	rFlodesDifferensMellanMinOchMax : REAL;
	rFlodesHojning1 : REAL; // Flödeshöjning uträknat.
	rFlodesHojning2 : REAL; // Flödeshöjning uträknat.
	rFlodesHojning3 : REAL; // Flödeshöjning uträknat.
	rFlodesHojning4 : REAL; // Flödeshöjning uträknat.
	rFlodesHojning5 : REAL; // Flödeshöjning uträknat.
	rFlodesHojning6 : REAL; // Flödeshöjning uträknat.
	rFlodesHojning7 : REAL; // Flödeshöjning uträknat.
	rFlodesHojning8 : REAL; // Flödeshöjning uträknat.
	rFlodesHojning9 : REAL; // Flödeshöjning uträknat.
	rFlodesHojning10 : REAL; // Flödeshöjning uträknat.
	rFlodesHojning11 : REAL; // Flödeshöjning uträknat.
	rFlodesHojning12 : REAL; // Flödeshöjning uträknat.
	rFlodesHojning13: REAL; // Flödeshöjning uträknat.
	rFlodesHojning14 : REAL; // Flödeshöjning uträknat.
	rFlodesHojning15 : REAL; // Flödeshöjning uträknat.
	rOmraknadFlodeskompenseringsSignal1 : REAL; // Flödeskompenseringsinput omräknad till 0-100 värde.
	rOmraknadFlodeskompenseringsSignal2 : REAL; // Flödeskompenseringsinput omräknad till 0-100 värde.
	rOmraknadFlodeskompenseringsSignal3 : REAL; // Flödeskompenseringsinput omräknad till 0-100 värde.
	rOmraknadFlodeskompenseringsSignal4 : REAL; // Flödeskompenseringsinput omräknad till 0-100 värde.
	rOmraknadFlodeskompenseringsSignal5 : REAL; // Flödeskompenseringsinput omräknad till 0-100 värde.
	rOmraknadFlodeskompenseringsSignal6 : REAL; // Flödeskompenseringsinput omräknad till 0-100 värde.
	rOmraknadFlodeskompenseringsSignal7 : REAL; // Flödeskompenseringsinput omräknad till 0-100 värde.
	rOmraknadFlodeskompenseringsSignal8 : REAL; // Flödeskompenseringsinput omräknad till 0-100 värde.
	rOmraknadFlodeskompenseringsSignal9 : REAL; // Flödeskompenseringsinput omräknad till 0-100 värde.
	rOmraknadFlodeskompenseringsSignal10 : REAL; // Flödeskompenseringsinput omräknad till 0-100 värde.
	rOmraknadFlodeskompenseringsSignal11 : REAL; // Flödeskompenseringsinput omräknad till 0-100 värde.
	rOmraknadFlodeskompenseringsSignal12 : REAL; // Flödeskompenseringsinput omräknad till 0-100 värde.
	rOmraknadFlodeskompenseringsSignal13 : REAL; // Flödeskompenseringsinput omräknad till 0-100 värde.
	rOmraknadFlodeskompenseringsSignal14 : REAL; // Flödeskompenseringsinput omräknad till 0-100 värde.
	rOmraknadFlodeskompenseringsSignal15 : REAL; // Flödeskompenseringsinput omräknad till 0-100 värde.
	bSekvensFlagga : BOOL;
	wResetConfirmed : WORD;
	
	fbSetpointConfirmed : FB_MBReadRegs;
	fbWriteSetpoint: FB_MBWriteSingleReg;
	rFlowSetpoint : REAL;
	wFlowSetpoint : WORD;
	wFlowSetpointConfirmed : WORD;
	bExecute1 : BOOL;
	wFlow : WORD;
	wOperationPoint : WORD;
	
	fbDamperPosition : FB_MBReadRegs;

	
	fbProcessValue : FB_MBReadRegs;
			
	fbReadValues : FB_MBReadRegs;
	
	fbOperationModeConfirmed : FB_MBReadRegs;
	fbWriteOperationMode: FB_MBWriteSingleReg;
	wOperationModeConfirmed : WORD;
	
	fbModeConfirmed : FB_MBReadRegs;
	fbWriteMode: FB_MBWriteSingleReg;
	wModeConfirmed : WORD;
	
	bExecute2 : BOOL;
	bExecute3 : BOOL;
	bExecute4 : BOOL;

	fbDoubleControlledModbusHoldingMinFlow,fbDoubleControlledModbusHoldingMaxFlow: fbDoubleControlledModbusHolding;
	fbHoldingRead : FB_MBReadRegs;
	
	rTemp : REAL; 
	sIP: STRING(255);
	sPort: STRING(255);
	sModbusID: STRING(255);
	sModbusLoop: STRING(255);
	sTemp: STRING(255);
	
	wWtest : WORD;
	
	rMid : REAL;
	
	//Kommunikationsfel
	fbKommTof : tof; 
	fbKommTon : ton;
END_VAR
VAR_INPUT PERSISTENT
	M AT %M*  : BOOL; // Manuellt läge börvärde~wp:
	OPM AT %M*  : REAL; // Manuellt börvärde~wp:[unit]%[format]0
END_VAR

//Modbus konfiguering
	sIP := CONCAT (SIPAddr, '');
	sPort := CONCAT ('<br>Port: ', UINT_TO_STRING(nTCPPort)); 								
	sModbusID := CONCAT('<br>ID: ', UINT_TO_STRING(nUnitID));
	sModbusLoop := CONCAT('<br>Loop: ', INT_TO_STRING(nModbusLoop));
	sTemp := sIP;
	sTemp := CONCAT(sTemp, sPort);
	sTemp := CONCAT(sTemp, sModbusID);
	sTemp := CONCAT(sTemp, sModbusLoop);
	PV8 := sTemp;

	bSekvensFlagga := oaksGVL.aBModbusSekvens[nModbusLoop] = UINT_TO_INT(nUnitID);
	//fbTp01(IN:=oaksGVL.aBModbusSekvens[nModbusLoop] = UINT_TO_INT(nUnitID) , PT:=T#5S , Q=> , ET=> );
	
	rFlodesDifferensMellanMinOchMax := SP2 - SP1;
	rOmraknadFlodeskompenseringsSignal1 := fScale2pInternalSetpoint(rX:=rFlodesHojning1 , Y1:=0 , Y2:=100 , X1:=0 , X2:=rFlodesDifferensMellanMinOchMax ); // Räknar om flödeskompenseringssignal till 0-100 värde.
	rOmraknadFlodeskompenseringsSignal2 := fScale2pInternalSetpoint(rX:=rFlodesHojning2 , Y1:=0 , Y2:=100 , X1:=0 , X2:=rFlodesDifferensMellanMinOchMax ); // Räknar om flödeskompenseringssignal till 0-100 värde.
	rOmraknadFlodeskompenseringsSignal3 := fScale2pInternalSetpoint(rX:=rFlodesHojning3 , Y1:=0 , Y2:=100 , X1:=0 , X2:=rFlodesDifferensMellanMinOchMax ); // Räknar om flödeskompenseringssignal till 0-100 värde.
	rOmraknadFlodeskompenseringsSignal4 := fScale2pInternalSetpoint(rX:=rFlodesHojning4 , Y1:=0 , Y2:=100 , X1:=0 , X2:=rFlodesDifferensMellanMinOchMax ); // Räknar om flödeskompenseringssignal till 0-100 värde.
	rOmraknadFlodeskompenseringsSignal5 := fScale2pInternalSetpoint(rX:=rFlodesHojning5 , Y1:=0 , Y2:=100 , X1:=0 , X2:=rFlodesDifferensMellanMinOchMax ); // Räknar om flödeskompenseringssignal till 0-100 värde.
	rOmraknadFlodeskompenseringsSignal6 := fScale2pInternalSetpoint(rX:=rFlodesHojning6 , Y1:=0 , Y2:=100 , X1:=0 , X2:=rFlodesDifferensMellanMinOchMax ); // Räknar om flödeskompenseringssignal till 0-100 värde.
	rOmraknadFlodeskompenseringsSignal7 := fScale2pInternalSetpoint(rX:=rFlodesHojning7 , Y1:=0 , Y2:=100 , X1:=0 , X2:=rFlodesDifferensMellanMinOchMax ); // Räknar om flödeskompenseringssignal till 0-100 värde.
	
	rOmraknadFlodeskompenseringsSignal8 := fScale2pInternalSetpoint(rX:=rFlodesHojning8 , Y1:=0 , Y2:=100 , X1:=0 , X2:=rFlodesDifferensMellanMinOchMax ); // Räknar om flödeskompenseringssignal till 0-100 värde.
	rOmraknadFlodeskompenseringsSignal9 := fScale2pInternalSetpoint(rX:=rFlodesHojning9 , Y1:=0 , Y2:=100 , X1:=0 , X2:=rFlodesDifferensMellanMinOchMax ); // Räknar om flödeskompenseringssignal till 0-100 värde.
	rOmraknadFlodeskompenseringsSignal10 := fScale2pInternalSetpoint(rX:=rFlodesHojning10 , Y1:=0 , Y2:=100 , X1:=0 , X2:=rFlodesDifferensMellanMinOchMax ); // Räknar om flödeskompenseringssignal till 0-100 värde.
	rOmraknadFlodeskompenseringsSignal11 := fScale2pInternalSetpoint(rX:=rFlodesHojning11 , Y1:=0 , Y2:=100 , X1:=0 , X2:=rFlodesDifferensMellanMinOchMax ); // Räknar om flödeskompenseringssignal till 0-100 värde.
	rOmraknadFlodeskompenseringsSignal12 := fScale2pInternalSetpoint(rX:=rFlodesHojning12 , Y1:=0 , Y2:=100 , X1:=0 , X2:=rFlodesDifferensMellanMinOchMax ); // Räknar om flödeskompenseringssignal till 0-100 värde.
	rOmraknadFlodeskompenseringsSignal13 := fScale2pInternalSetpoint(rX:=rFlodesHojning13 , Y1:=0 , Y2:=100 , X1:=0 , X2:=rFlodesDifferensMellanMinOchMax ); // Räknar om flödeskompenseringssignal till 0-100 värde.
	rOmraknadFlodeskompenseringsSignal14 := fScale2pInternalSetpoint(rX:=rFlodesHojning14 , Y1:=0 , Y2:=100 , X1:=0 , X2:=rFlodesDifferensMellanMinOchMax ); // Räknar om flödeskompenseringssignal till 0-100 värde.
	rOmraknadFlodeskompenseringsSignal15 := fScale2pInternalSetpoint(rX:=rFlodesHojning15 , Y1:=0 , Y2:=100 , X1:=0 , X2:=rFlodesDifferensMellanMinOchMax ); // Räknar om flödeskompenseringssignal till 0-100 värde.
(*
	Börvärde 0 WORD 0…10000 r/w Börvärde [%] 0=0%, 10000=100%
	se adress 122:
	'0': Börvärde är endast läsvärde
*)	
	IF M  THEN
		PV4 := OPM;
	ELSIF bFlodesBalanseringAktiv THEN
		PV4 := rFlodesBalansering;
	ELSE
		PV4 := rSetpoint + rOmraknadFlodeskompenseringsSignal1+rOmraknadFlodeskompenseringsSignal2+rOmraknadFlodeskompenseringsSignal3+rOmraknadFlodeskompenseringsSignal4+rOmraknadFlodeskompenseringsSignal5
		+rOmraknadFlodeskompenseringsSignal6+rOmraknadFlodeskompenseringsSignal7+rOmraknadFlodeskompenseringsSignal8+rOmraknadFlodeskompenseringsSignal9+rOmraknadFlodeskompenseringsSignal10
		+rOmraknadFlodeskompenseringsSignal11+rOmraknadFlodeskompenseringsSignal12+rOmraknadFlodeskompenseringsSignal13+rOmraknadFlodeskompenseringsSignal14+rOmraknadFlodeskompenseringsSignal15; 
	END_IF
	
	AL8 := M;

	
	rFlowSetpoint := fScale2pInternalSetpoint(rX:=PV4 , Y1:=0 , Y2:=10000 , X1:=0 , X2:= 100);

	

	
(**** RESET START ****)
	IF fHyst(rProcessValue :=rFlowSetpoint ,rSetPoint:=REAL_TO_WORD(wFlowSetpointConfirmed) ,rDevLimit:=10) AND wOperationModeInternal = 1 THEN
		wFlowSetpoint := REAL_TO_WORD(rFlowSetpoint);
		bExecute1 := TRUE;
	ELSE
		bExecute1 := FALSE;
	END_IF;

	fbWriteSetpoint(
	sIPAddr:= sIpAddr, 
	nTCPPort:= INT_TO_UINT(nTCPPort), 
	nUnitID:= INT_TO_BYTE(nUnitID), 
	nMBAddr:= 0, 
	nValue:= wFlowSetpoint, 
	bExecute:= bExecute1 AND bSekvensFlagga, 
	tTimeout:=T#20S , 
	bBusy=> , 
	bError=> , 
	nErrId=> );
	
	fbSetpointConfirmed(
	sIPAddr:= sIpAddr, 
	nTCPPort:= INT_TO_UINT(nTCPPort), 
	nUnitID:= INT_TO_BYTE(nUnitID), 
	nQuantity:= 1, 
	nMBAddr:= 0, 
	cbLength:= SIZEOF(wFlowSetpointConfirmed), 
	pDestAddr:= ADR(wFlowSetpointConfirmed), 
	bExecute:= bSekvensFlagga, 
	tTimeout:= T#20S, 
	cbRead=> );
(**** Spjällposition ****)
	fbDamperPosition(
	sIPAddr:= sIpAddr, 
	nTCPPort:= INT_TO_UINT(nTCPPort), 
	nUnitID:= INT_TO_BYTE(nUnitID), 
	nQuantity:= 1, 
	nMBAddr:= 4, 
	cbLength:= SIZEOF(wOperationPoint), 
	pDestAddr:= ADR(wOperationPoint), 
	bExecute:= bSekvensFlagga, 
	tTimeout:= T#20S, 
	cbRead=> );
	OP := WORD_TO_REAL(wOperationPoint) /100.0;
	
(* Ärvärde flöde *) 
	fbProcessValue(
	sIPAddr:= sIpAddr, 
	nTCPPort:= INT_TO_UINT(nTCPPort), 
	nUnitID:= INT_TO_BYTE(nUnitID), 
	nQuantity:= 1, 
	nMBAddr:= 7, 
	cbLength:= SIZEOF(wFlow), 
	pDestAddr:= ADR(wFlow), 
	bExecute:= bSekvensFlagga, 
	tTimeout:= T#20S, 
	cbRead=> );
	PV := WORD_TO_REAL(wFlow);
(* Kollar så att spjäll är i rätt driftläge *)	
	fbOperationModeConfirmed(
	sIPAddr:= sIpAddr, 
	nTCPPort:= INT_TO_UINT(nTCPPort), 
	nUnitID:= INT_TO_BYTE(nUnitID), 
	nQuantity:= 1, 
	nMBAddr:= 122, 
	cbLength:= SIZEOF(wOperationModeConfirmed), 
	pDestAddr:= ADR(wOperationModeConfirmed), 
	bExecute:= bSekvensFlagga, 
	tTimeout:= T#20S, 
	cbRead=> );
	
	wOperationModeInternal := mOperationMode(M,wOperationMode);
	
	IF wOperationModeInternal <> wOperationModeConfirmed THEN
		bExecute2 := TRUE;
	ELSE
		bExecute2 := FALSE;
	END_IF;
	fbWriteOperationMode(
	sIPAddr:= sIpAddr, 
	nTCPPort:= INT_TO_UINT(nTCPPort), 
	nUnitID:= INT_TO_BYTE(nUnitID), 
	nMBAddr:= 122, 
	nValue:= wOperationModeInternal, 
	bExecute:= bExecute2 AND bSekvensFlagga , 
	tTimeout:=T#20S , 
	bBusy=> , 
	bError=> , 
	nErrId=> );
	
	
	fbHoldingRead(
	sIPAddr:= sIpAddr, 
	nTCPPort:= INT_TO_UINT(nTCPPort), 
	nUnitID:= INT_TO_BYTE(nUnitID), 
	nMBAddr:= 120, 
	nQuantity:=1 , 
	cbLength:= SIZEOF(wWtest), 
	pDestAddr:=ADR(wWtest) , 
	bExecute:=bSekvensFlagga , 
	tTimeout:=T#20S , 
	bBusy=> , 
	bError=> , 
	nErrId=> , 
	cbRead=> );
	
	fbDoubleControlledModbusHoldingMinFlow(
	sIPAddr:= sIpAddr, 
	nTCPPort:= INT_TO_UINT(nTCPPort), 
	nUnitID:= INT_TO_BYTE(nUnitID), 
	nMBAddr:= 120, 
	tTimeout:=T#20S,
	tStartDelay:=T#0MS,
	bExecute:=bSekvensFlagga, 
	rScale:=1 , 
	rWrite:= SP1, 
	bBusy=> , 
	bError=> );
	
	fbDoubleControlledModbusHoldingMaxFlow(
	sIPAddr:= sIpAddr, 
	nTCPPort:= INT_TO_UINT(nTCPPort), 
	nUnitID:= INT_TO_BYTE(nUnitID), 
	nMBAddr:= 121, 
	tTimeout:=T#20S,
	tStartDelay:=T#100MS ,
	bExecute:=bSekvensFlagga, 
	rScale:=1 , 
	rWrite:= SP2, 
	bBusy=> , 
	bError=> );

	//Skriver driftläge
	IF wMode <> wModeConfirmed THEN
		bExecute4 := TRUE;
	ELSE
		bExecute4 := FALSE;
	END_IF;
	
	fbWriteMode(
	sIPAddr:= sIpAddr, 
	nTCPPort:= INT_TO_UINT(nTCPPort), 
	nUnitID:= INT_TO_BYTE(nUnitID), 
	nMBAddr:= 1, 
	nValue:= wMode, 
	bExecute:= bExecute4 AND bSekvensFlagga AND bMode, 
	tTimeout:=T#20S , 
	bBusy=> , 
	bError=> , 
	nErrId=> );
	
	fbModeConfirmed(
	sIPAddr:= sIpAddr, 
	nTCPPort:= INT_TO_UINT(nTCPPort), 
	nUnitID:= INT_TO_BYTE(nUnitID), 
	nQuantity:= 1, 
	nMBAddr:= 1, 
	cbLength:= SIZEOF(wModeConfirmed), 
	pDestAddr:= ADR(wModeConfirmed), 
	bExecute:= bSekvensFlagga, 
	tTimeout:= T#20S, 
	cbRead=> );	
	
	// Räknar ut aktuellt börvärde
	rTemp := WORD_TO_REAL(wFlowSetpointConfirmed);
	rMid := 5000;
	IF 	  wMode = 0 THEN
		  CSP := OaksLibrary.fScale2pInternalSetpoint(rX:=rTemp , Y1:=SP1 , Y2:=SP2 , X1:=0 , X2:=10000 );
	ELSIF wMode = 1 THEN
		  CSP := SP2;
	ELSIF wMode = 2 THEN
		  CSP := 0;
	ELSIF wMode = 3 THEN 
		  CSP := SP1;
	ELSIF wMode = 4 THEN
		  CSP := SP2;
	ELSIF wMode = 5 THEN
		  CSP :=OaksLibrary.fScale2pInternalSetpoint(rX:=rMid , Y1:=SP1 , Y2:=SP2 , X1:=0 , X2:=10000 );
	END_IF
	
	oaksGVL.aBModbusBusyFlagga[nModbusLoop,nUnitID] := fbProcessValue.bBusy OR fbWriteSetpoint.bBusy OR fbDamperPosition.bBusy OR fbSetpointConfirmed.bBusy
	OR fbWriteOperationMode.bBusy OR fbOperationModeConfirmed.bBusy OR fbDoubleControlledModbusHoldingMinFlow.bBusy OR fbDoubleControlledModbusHoldingMaxFlow.bBusy OR fbWriteMode.bBusy OR fbModeConfirmed.bBusy;// OR fbTp01.Q;
	
//Communication error
	PV7 := NOT fbKommTof.Q;
	fbKommTof(IN:=fbProcessValue.bError , PT:=T#20S , Q=> , ET=> );
	fbKommTon(IN:=fbKommTof.Q , PT:=T#20M , Q=> , ET=> );
	FAULT :=fbKommTon.Q;

// Metod för att balansera flöde så att spjäll får samma som anges här. Används denna metod struntar blocket i inputen rSetpoint.
METHOD PUBLIC mFlodesBalansering
VAR_INPUT
	rBalanseratFlode : REAL;
END_VAR
rFlodesBalansering := fScale2pInternalSetpoint(rBalanseratFlode,0,100,SP1,SP2);
bFlodesBalanseringAktiv := TRUE;
END_METHOD

METHOD PUBLIC mFlodesKompensering1
VAR_IN_OUT
	fbSwegonReact01 : fbSwegonReact;
END_VAR
rFlodesHojning1 :=  fbSwegonReact01.CSP - fbSwegonReact01.SP1;
END_METHOD

METHOD PUBLIC mFlodesKompensering10
VAR_IN_OUT
	fbSwegonReact10 : fbSwegonReact;
END_VAR
rFlodesHojning10 :=  fbSwegonReact10.CSP - fbSwegonReact10.SP1;
END_METHOD

METHOD PUBLIC mFlodesKompensering11
VAR_IN_OUT
	fbSwegonReact11 : fbSwegonReact;
END_VAR
rFlodesHojning11 :=  fbSwegonReact11.CSP - fbSwegonReact11.SP1;
END_METHOD

METHOD PUBLIC mFlodesKompensering12
VAR_IN_OUT
	fbSwegonReact12 : fbSwegonReact;
END_VAR
rFlodesHojning12 :=  fbSwegonReact12.CSP - fbSwegonReact12.SP1;
END_METHOD

METHOD PUBLIC mFlodesKompensering13
VAR_IN_OUT
	fbSwegonReact13 : fbSwegonReact;
END_VAR
rFlodesHojning13 :=  fbSwegonReact13.CSP - fbSwegonReact13.SP1;
END_METHOD

METHOD PUBLIC mFlodesKompensering14
VAR_IN_OUT
	fbSwegonReact14 : fbSwegonReact;
END_VAR
rFlodesHojning14 :=  fbSwegonReact14.CSP - fbSwegonReact14.SP1;
END_METHOD

METHOD PUBLIC mFlodesKompensering15
VAR_IN_OUT
	fbSwegonReact15 : fbSwegonReact;
END_VAR
rFlodesHojning15 :=  fbSwegonReact15.CSP - fbSwegonReact15.SP1;
END_METHOD

METHOD PUBLIC mFlodesKompensering2
VAR_IN_OUT
	fbSwegonReact02 : fbSwegonReact;
END_VAR
rFlodesHojning2 :=  fbSwegonReact02.CSP - fbSwegonReact02.SP1;
END_METHOD

METHOD PUBLIC mFlodesKompensering3
VAR_IN_OUT
	fbSwegonReact03 : fbSwegonReact;
END_VAR
rFlodesHojning3 :=  fbSwegonReact03.CSP - fbSwegonReact03.SP1;
END_METHOD

METHOD PUBLIC mFlodesKompensering4
VAR_IN_OUT
	fbSwegonReact04 : fbSwegonReact;
END_VAR
rFlodesHojning4 :=  fbSwegonReact04.CSP - fbSwegonReact04.SP1;
END_METHOD

METHOD PUBLIC mFlodesKompensering5
VAR_IN_OUT
	fbSwegonReact05 : fbSwegonReact;
END_VAR
rFlodesHojning5 :=  fbSwegonReact05.CSP - fbSwegonReact05.SP1;
END_METHOD

METHOD PUBLIC mFlodesKompensering6
VAR_IN_OUT
	fbSwegonReact06 : fbSwegonReact;
END_VAR
rFlodesHojning6 :=  fbSwegonReact06.CSP - fbSwegonReact06.SP1;
END_METHOD

METHOD PUBLIC mFlodesKompensering7
VAR_IN_OUT
	fbSwegonReact07 : fbSwegonReact;
END_VAR
rFlodesHojning7 :=  fbSwegonReact07.CSP - fbSwegonReact07.SP1;
END_METHOD

METHOD PUBLIC mFlodesKompensering8
VAR_IN_OUT
	fbSwegonReact08 : fbSwegonReact;
END_VAR
rFlodesHojning8 :=  fbSwegonReact08.CSP - fbSwegonReact08.SP1;
END_METHOD

METHOD PUBLIC mFlodesKompensering9
VAR_IN_OUT
	fbSwegonReact09 : fbSwegonReact;
END_VAR
rFlodesHojning9 :=  fbSwegonReact09.CSP - fbSwegonReact09.SP1;
END_METHOD

METHOD PRIVATE mOperationMode : WORD
VAR_INPUT
	M : BOOL;
	wOperationMode : WORD;
END_VAR
IF M THEN
	mOperationMode := 1;
ELSE
	mOperationMode := wOperationMode;
END_IF
END_METHOD

END_FUNCTION_BLOCK

// oaksModbusLibrary/Swegon/fbSwegonReactPx
//OAKS AB
//2020-11-18
//Funktionsblock för kommunikation med Swegon React PX (tryckreglerat spjäll)
//Dubbelriktad modbusskrivning för börvärde
FUNCTION_BLOCK fbSwegonReactPx
VAR_INPUT
	sIPAddr : STRING := ''; 
	nTCPPort : UINT;
	nUnitID : UINT;
	nModbusLoop : UINT := 1;
	rSetpoint : REAL; // Trycksignal mellan 0-100
	wOperationMode : WORD := 1; // Driftläge (0 = börvärde via analog in 0-10V, 1 = börvärde via modbus)
	wMode : WORD := 0; //Överstyrning spjälläge 0: None 1: Open 2: Close 3: Min 4: Max 5: Mid
	wBusErrorMode : WORD := 0; // Position vid kommunikationsbortfall 120s 0=Ej aktivt, 1=Spjäll stänger, 2=Spjäll öppnar 
	SP1 AT %M*  : REAL; //Inställt min. tryck~wp:[unit]Pa[format]0
	SP2 AT %M*  : REAL; //Inställt max. tryck~wp:[unit]Pa[format]0

END_VAR
VAR_OUTPUT
	CSP AT %M*  : REAL; //Aktuellt börvärde~wp:[trendoption]i:300[unit]Pa[format]0
	OP AT %M*  : REAL; //Spjällposition relativ~wp:[trendoption]i:300[unit]%[format]0
	PV4 AT %M*  : REAL; //Uträknat börvärde~wp:[trendoption]i:300[unit]%[format]0
	AL8 AT %M*  : BOOL; //Handställningslarm~wp:
	PV AT %M*  : REAL; //Ärvärde tryck~wp:[trendoption]i:300[unit]Pa[format]0
	PV7 AT %M* : BOOL;//Senaste läsning OK~wp:
	PV8 AT %M* : STRING;//Modbus konfiguering~wp:
	FAULT AT %M* : BOOL;//Kommunikationsfel~wp:
END_VAR
VAR
	bSekvensFlagga : BOOL;
	wResetConfirmed : WORD;
	
	fbSetpointConfirmed : FB_MBReadRegs;
	fbWriteSetpoint: FB_MBWriteSingleReg;
	rPressureSetpoint : REAL;
	wPressureSetpoint : WORD;
	wPressureSetpointConfirmed : WORD;
	bExecute1 : BOOL;
	wPressure : WORD;
	wOperationPoint : WORD;
	
	fbDamperPosition : FB_MBReadRegs;
	fbProcessValue : FB_MBReadRegs;
	fbReadValues : FB_MBReadRegs;
		
	fbOperationModeConfirmed : FB_MBReadRegs;
	fbWriteOperationMode: FB_MBWriteSingleReg;
	wOperationModeConfirmed : WORD;
	bExecute2 : BOOL;
	bExecute3 : BOOL;
	bExecute4 : BOOL;
	
	fbModeConfirmed : FB_MBReadRegs;
	fbWriteMode: FB_MBWriteSingleReg;
	wModeConfirmed : WORD;
	
	fbDoubleControlledModbusHoldingMinPressure,fbDoubleControlledModbusHoldingMaxPressure: fbDoubleControlledModbusHolding;
	fbHoldingRead : FB_MBReadRegs;
	rTemp : REAL; 
	sIP: STRING(255);
	sPort: STRING(255);
	sModbusID: STRING(255);
	sModbusLoop: STRING(255);
	sTemp: STRING(255);
	
	wWtest : WORD;
	
	//Läge vid kommunikationsfel
	fbWriteBusErrorModeConfirmed : FB_MBReadRegs;
	fbWriteBusErrorMode: FB_MBWriteSingleReg;
	wWriteBusErrorModeConfirmed : WORD;
	
	//Kommunikationsfel
	fbKommTof : tof; 
	fbKommTon : ton;
END_VAR
VAR_INPUT PERSISTENT
	M AT %M*  : BOOL; // Manuellt läge börvärde~wp:
	OPM AT %M*  : REAL; // Manuellt börvärde~wp:[unit]%[format]0
END_VAR

//Modbus konfiguering
	sIP := CONCAT (SIPAddr, '');
	sPort := CONCAT ('<br>Port: ', UINT_TO_STRING(nTCPPort)); 								
	sModbusID := CONCAT('<br>ID: ', UINT_TO_STRING(nUnitID));
	sModbusLoop := CONCAT('<br>Loop: ', INT_TO_STRING(nModbusLoop));
	sTemp := sIP;
	sTemp := CONCAT(sTemp, sPort);
	sTemp := CONCAT(sTemp, sModbusID);
	sTemp := CONCAT(sTemp, sModbusLoop);
	PV8 := sTemp;

	bSekvensFlagga := oaksGVL.aBModbusSekvens[nModbusLoop] = UINT_TO_INT(nUnitID);

//Manuellt börvärde	
	IF M  THEN
		PV4 := OPM; 
	ELSE
		PV4 := rSetpoint;  
	END_IF
	
	AL8 := M;
	
	rPressureSetpoint := fScale2pInternalSetpoint(rX:=PV4 , Y1:=0 , Y2:=10000 , X1:=0 , X2:= 100);
	
	fbHoldingRead(
	sIPAddr:= sIpAddr, 
	nTCPPort:= INT_TO_UINT(nTCPPort), 
	nUnitID:= INT_TO_BYTE(nUnitID), 
	nMBAddr:= 120, 
	nQuantity:=1 , 
	cbLength:= SIZEOF(wWtest), 
	pDestAddr:=ADR(wWtest) , 
	bExecute:=bSekvensFlagga , 
	tTimeout:=T#20S , 
	bBusy=> , 
	bError=> , 
	nErrId=> , 
	cbRead=> );
	
	fbDoubleControlledModbusHoldingMinPressure(
	sIPAddr:= sIpAddr, 
	nTCPPort:= INT_TO_UINT(nTCPPort), 
	nUnitID:= INT_TO_BYTE(nUnitID), 
	nMBAddr:= 120, 
	tTimeout:=T#20S,
	tStartDelay:=T#0MS,
	bExecute:=bSekvensFlagga, 
	rScale:=1 , 
	rWrite:= SP1, 
	bBusy=> , 
	bError=> );
	
	fbDoubleControlledModbusHoldingMaxPressure(
	sIPAddr:= sIpAddr, 
	nTCPPort:= INT_TO_UINT(nTCPPort), 
	nUnitID:= INT_TO_BYTE(nUnitID), 
	nMBAddr:= 121, 
	tTimeout:=T#20S,
	tStartDelay:=T#0MS ,
	bExecute:=bSekvensFlagga, 
	rScale:=1 , 
	rWrite:= SP2, 
	bBusy=> , 
	bError=> );
	
(**** RESET START ****)
	IF fHyst(rProcessValue :=rPressureSetpoint ,rSetPoint:=REAL_TO_WORD(wPressureSetpointConfirmed) ,rDevLimit:=10) AND wOperationMode = 1 THEN
		wPressureSetpoint := REAL_TO_WORD(rPressureSetpoint);
		bExecute1 := TRUE;
	ELSE
		bExecute1 := FALSE;
	END_IF;

	fbWriteSetpoint(
	sIPAddr:= sIpAddr, 
	nTCPPort:= INT_TO_UINT(nTCPPort), 
	nUnitID:= INT_TO_BYTE(nUnitID), 
	nMBAddr:= 0, 
	nValue:= wPressureSetpoint, 
	bExecute:= bExecute1 AND bSekvensFlagga, 
	tTimeout:=T#20S , 
	bBusy=> , 
	bError=> , 
	nErrId=> );
	
	fbSetpointConfirmed(
	sIPAddr:= sIpAddr, 
	nTCPPort:= INT_TO_UINT(nTCPPort), 
	nUnitID:= INT_TO_BYTE(nUnitID), 
	nQuantity:= 1, 
	nMBAddr:= 0, 
	cbLength:= SIZEOF(wPressureSetpointConfirmed), 
	pDestAddr:= ADR(wPressureSetpointConfirmed), 
	bExecute:= bSekvensFlagga, 
	tTimeout:= T#20S, 
	cbRead=> );
(**** Spjällposition ****)
	fbDamperPosition(
	sIPAddr:= sIpAddr, 
	nTCPPort:= INT_TO_UINT(nTCPPort), 
	nUnitID:= INT_TO_BYTE(nUnitID), 
	nQuantity:= 1, 
	nMBAddr:= 4, 
	cbLength:= SIZEOF(wOperationPoint), 
	pDestAddr:= ADR(wOperationPoint), 
	bExecute:= bSekvensFlagga, 
	tTimeout:= T#20S, 
	cbRead=> );
	OP := WORD_TO_REAL(wOperationPoint) /100.0;
(* Ärvärde tryck *) 
	fbProcessValue(
	sIPAddr:= sIpAddr, 
	nTCPPort:= INT_TO_UINT(nTCPPort), 
	nUnitID:= INT_TO_BYTE(nUnitID), 
	nQuantity:= 1, 
	nMBAddr:= 7, 
	cbLength:= SIZEOF(wPressure), 
	pDestAddr:= ADR(wPressure), 
	bExecute:= bSekvensFlagga, 
	tTimeout:= T#20S, 
	cbRead=> );
	PV := WORD_TO_REAL(wPressure);
(* Kollar så att spjäll är i rätt driftläge *)	
	IF wOperationMode <> wOperationModeConfirmed THEN
		bExecute2 := TRUE;
	ELSE
		bExecute2 := FALSE;
	END_IF;
	fbWriteOperationMode(
	sIPAddr:= sIpAddr, 
	nTCPPort:= INT_TO_UINT(nTCPPort), 
	nUnitID:= INT_TO_BYTE(nUnitID), 
	nMBAddr:= 122, 
	nValue:= wOperationMode, 
	bExecute:= bExecute2 AND bSekvensFlagga, 
	tTimeout:=T#20S , 
	bBusy=> , 
	bError=> , 
	nErrId=> );
	
	fbOperationModeConfirmed(
	sIPAddr:= sIpAddr, 
	nTCPPort:= INT_TO_UINT(nTCPPort), 
	nUnitID:= INT_TO_BYTE(nUnitID), 
	nQuantity:= 1, 
	nMBAddr:= 122, 
	cbLength:= SIZEOF(wOperationModeConfirmed), 
	pDestAddr:= ADR(wOperationModeConfirmed), 
	bExecute:= bSekvensFlagga, 
	tTimeout:= T#20S, 
	cbRead=> );
	
//Ställer in läge vid kommunikationsfelslarm
	IF wBusErrorMode <> wWriteBusErrorModeConfirmed THEN
		bExecute3 := TRUE;
	ELSE
		bExecute3 := FALSE;
	END_IF;
	fbWriteBusErrorMode(
	sIPAddr:= sIpAddr, 
	nTCPPort:= INT_TO_UINT(nTCPPort), 
	nUnitID:= INT_TO_BYTE(nUnitID), 
	nMBAddr:= 108, 
	nValue:= wBusErrorMode, 
	bExecute:= bExecute3 AND bSekvensFlagga, 
	tTimeout:=T#20S , 
	bBusy=> , 
	bError=> , 
	nErrId=> );
	
	fbWriteBusErrorModeConfirmed(
	sIPAddr:= sIpAddr, 
	nTCPPort:= INT_TO_UINT(nTCPPort), 
	nUnitID:= INT_TO_BYTE(nUnitID), 
	nQuantity:= 1, 
	nMBAddr:= 108, 
	cbLength:= SIZEOF(wWriteBusErrorModeConfirmed), 
	pDestAddr:= ADR(wWriteBusErrorModeConfirmed), 
	bExecute:= bSekvensFlagga, 
	tTimeout:= T#20S, 
	cbRead=> );
	
//Skriver driftläge
	IF wMode <> wModeConfirmed THEN
		bExecute4 := TRUE;
	ELSE
		bExecute4 := FALSE;
	END_IF;
	
	fbWriteMode(
	sIPAddr:= sIpAddr, 
	nTCPPort:= INT_TO_UINT(nTCPPort), 
	nUnitID:= INT_TO_BYTE(nUnitID), 
	nMBAddr:= 1, 
	nValue:= wMode, 
	bExecute:= bExecute4 AND bSekvensFlagga, 
	tTimeout:=T#20S , 
	bBusy=> , 
	bError=> , 
	nErrId=> );
	
	fbModeConfirmed(
	sIPAddr:= sIpAddr, 
	nTCPPort:= INT_TO_UINT(nTCPPort), 
	nUnitID:= INT_TO_BYTE(nUnitID), 
	nQuantity:= 1, 
	nMBAddr:= 1, 
	cbLength:= SIZEOF(wModeConfirmed), 
	pDestAddr:= ADR(wModeConfirmed), 
	bExecute:= bSekvensFlagga, 
	tTimeout:= T#20S, 
	cbRead=> );	
	
//Räknar ut aktuellt börvärde
	rTemp := WORD_TO_REAL(wPressureSetpointConfirmed);
	CSP := OaksLibrary.fScale2pInternalSetpoint(rX:=rTemp , Y1:=SP1 , Y2:=SP2 , X1:=0 , X2:=10000 );
	
	oaksGVL.aBModbusBusyFlagga[nModbusLoop,nUnitID] := fbProcessValue.bBusy OR fbWriteSetpoint.bBusy OR fbDamperPosition.bBusy OR fbSetpointConfirmed.bBusy
	OR fbWriteOperationMode.bBusy OR fbOperationModeConfirmed.bBusy OR fbDoubleControlledModbusHoldingMinPressure.bBusy OR fbDoubleControlledModbusHoldingMaxPressure.bBusy OR fbWriteBusErrorModeConfirmed.bBusy OR fbWriteBusErrorMode.bBusy OR fbWriteMode.bBusy;
	
//Communication error
	PV7 := NOT fbKommTof.Q;
	fbKommTof(IN:=fbProcessValue.bError , PT:=T#20S , Q=> , ET=> );
	fbKommTon(IN:=fbKommTof.Q , PT:=T#20M , Q=> , ET=> );
	FAULT :=fbKommTon.Q;

END_FUNCTION_BLOCK

// oaksModbusLibrary/Swegon/fbSwegonWiseMasterSlave
//OAKS AB
//2020-05-12
//Grundfil för modbusblock
FUNCTION_BLOCK fbSwegonWiseMasterSlave
VAR_INPUT
	sIPAddr : STRING := ''; 
	nTCPPort : UINT;
	nUnitID : BYTE :=1;
	iModbusLoop : INT :=1; //Modbusslinga
	MASTERDAMPER_SP AT %M*  : REAL;  //Tilluftstryck~wp:[unit]Pa[format]0[trendoption]i:300
	SLAVEDAMPER_SP1 AT %M* : REAL;  //Frånluftsflöde offsett~wp:[unit]l/s[format]0[trendoption]i:300
END_VAR
VAR_OUTPUT
		
	PV8 AT %M* : STRING;//Modbus konfiguering~wp:
	MASTERDAMPER_FAULT AT %M*  : BOOL; //Kommunikationsfel Swegon Wise~wp:
	
	MASTERDAMPER_PV AT %M* : REAL;  //Tryck~wp:[unit]Pa[format]0[trendoption]i:300
	MASTERDAMPER_PV1 AT %M*  : REAL;  //Flöde~wp:[unit]l/s[format]0[trendoption]i:300
	MASTERDAMPER_OP AT %M*  : REAL;  //Spjällposition~wp:[unit]%[format]0[trendoption]i:300
	
	
	SLAVEDAMPER_OP AT %M*  : REAL;  //Spjällposition~wp:[unit]%[format]0[trendoption]i:300
	SLAVEDAMPER_PV1 AT %M*  : REAL;  //Flöde~wp:[unit]l/s[format]0[trendoption]i:300
	
END_VAR
VAR
	//Skrivning heat setpoint 
	FB_MBWriteSingleRegPressure: fbDoubleControlledModbusHolding;	
	FB_MBWriteSingleRegSlaveOffset: fbDoubleControlledModbusHolding;	
	
	FB_MBReadInputRegsSupPress : FB_MBReadInputRegs;
	wSupPress : WORD;	

	FB_MBReadInputRegsSupDamperPos : FB_MBReadInputRegs;
	wSupDamperPos : WORD;
	
	FB_MBReadInputRegsExhDamperPos : FB_MBReadInputRegs;
	wExhDamperPos : WORD;
	
	FB_MBReadInputRegsSupFlow : FB_MBReadInputRegs;
	wSupFlow : WORD;

	FB_MBReadInputRegsExhFlow : FB_MBReadInputRegs;
	wExhFlow : WORD;	


	offset : WORD;
	rTemp : REAL;
	iTemp : UINT;
	bSekvensFlagga : BOOL;
			

		
	//Kommunikationsfel
	fbKommTof : tof; 
	fbKommTon : ton;
	
	sIP: STRING(255);
	sPort: STRING(255);
	sModbusID: STRING(255);
	sModbusLoop: STRING(255);
	sTemp : STRING(255);
	
	
END_VAR

//General
	offset := 0;
//Sekvens	
	bSekvensFlagga := oaksGVL.aBModbusSekvens[iModbusLoop] = UINT_TO_INT(nUnitID);
//Modbus konfiguering
	sIP := CONCAT (SIPAddr, '');
	sPort := CONCAT ('<br>Port: ', UINT_TO_STRING(nTCPPort)); 								
	sModbusID := CONCAT('<br>ID: ', UINT_TO_STRING(nUnitID));
	sModbusLoop := CONCAT('<br>Loop: ', INT_TO_STRING(iModbusLoop));	

	sTemp := sIP;
	sTemp := CONCAT(sTemp, sPort);
	sTemp := CONCAT(sTemp, sModbusID);
	sTemp := CONCAT(sTemp, sModbusLoop);
	
	PV8 := sTemp;

///////////////		
//READ
///////////////		

	FB_MBReadInputRegsSupPress(
	sIPAddr:=sIPAddr, 
	nTCPPort:=nTCPPort , 
	nUnitID:=nUnitID , 
	nQuantity:= 1, 
	nMBAddr:= 56, 
	cbLength:= SIZEOF(wSupPress), 
	pDestAddr:= ADR(wSupPress), 
	bExecute:= bSekvensFlagga, 
	tTimeout:= , 
	bBusy=> , 
	bError=> , 
	nErrId=> , 
	cbRead=> );
	
	MASTERDAMPER_PV :=WORD_TO_REAL(wSupPress);

	FB_MBReadInputRegsSupDamperPos(
	sIPAddr:=sIPAddr, 
	nTCPPort:=nTCPPort , 
	nUnitID:=nUnitID , 
	nQuantity:= 1, 
	nMBAddr:= 54, 
	cbLength:= SIZEOF(wSupDamperPos), 
	pDestAddr:= ADR(wSupDamperPos), 
	bExecute:=bSekvensFlagga , 
	tTimeout:= , 
	bBusy=> , 
	bError=> , 
	nErrId=> , 
	cbRead=> );
	
	MASTERDAMPER_OP :=WORD_TO_REAL(wSupDamperPos);
	
	FB_MBReadInputRegsExhDamperPos(
	sIPAddr:=sIPAddr, 
	nTCPPort:=nTCPPort , 
	nUnitID:=nUnitID , 
	nQuantity:= 1, 
	nMBAddr:= 55, 
	cbLength:= SIZEOF(wExhDamperPos), 
	pDestAddr:= ADR(wExhDamperPos), 
	bExecute:= bSekvensFlagga, 
	tTimeout:= , 
	bBusy=> , 
	bError=> , 
	nErrId=> , 
	cbRead=> );
	
		
	SLAVEDAMPER_OP :=WORD_TO_REAL(wExhDamperPos);

	FB_MBReadInputRegsSupFlow(
	sIPAddr:=sIPAddr, 
	nTCPPort:=nTCPPort , 
	nUnitID:=nUnitID , 
	nQuantity:= 1, 
	nMBAddr:= 57, 
	cbLength:= SIZEOF(wSupFlow), 
	pDestAddr:= ADR(wSupFlow), 
	bExecute:= bSekvensFlagga, 
	tTimeout:= , 
	bBusy=> , 
	bError=> , 
	nErrId=> , 
	cbRead=> );
	
	MASTERDAMPER_PV1 :=WORD_TO_REAL(wSupFlow);
	
	
	FB_MBReadInputRegsExhFlow(
	sIPAddr:=sIPAddr, 
	nTCPPort:=nTCPPort , 
	nUnitID:=nUnitID , 
	nQuantity:= 1, 
	nMBAddr:= 58, 
	cbLength:= SIZEOF(wExhFlow), 
	pDestAddr:= ADR(wExhFlow), 
	bExecute:= bSekvensFlagga, 
	tTimeout:= , 
	bBusy=> , 
	bError=> , 
	nErrId=> , 
	cbRead=> );
	
	
	SLAVEDAMPER_PV1 :=WORD_TO_REAL(wExhFlow);
	
	FB_MBWriteSingleRegPressure(
	sIPAddr:=sIPAddr, 
	nTCPPort:=nTCPPort , 
	nUnitID:=nUnitID ,
	nMBAddr:= 35, 
	bExecute:=bSekvensFlagga , 
	rScale:= 1, 
	rWrite:=MASTERDAMPER_SP , 
	bBusy=> , 
	bError=> );
	
	FB_MBWriteSingleRegSlaveOffset(
	sIPAddr:=sIPAddr, 
	nTCPPort:=nTCPPort , 
	nUnitID:=nUnitID ,
	nMBAddr:=32 , 
	bExecute:=bSekvensFlagga , 
	rScale:= 1, 
	rWrite:= SLAVEDAMPER_SP1, 
	bBusy=> , 
	bError=> );
		
	
//Communication error
	fbKommTof(IN:=FB_MBReadInputRegsSupPress.bError , PT:=T#20S , Q=> , ET=> );
	fbKommTon(IN:=fbKommTof.Q , PT:=T#20M , Q=> , ET=> );
	MASTERDAMPER_FAULT :=fbKommTon.Q;
		
//Write busy	
	oaksgvl.aBModbusBusyFlagga[iModbusLoop,nUnitID] := FB_MBWriteSingleRegPressure.bBusy OR FB_MBWriteSingleRegSlaveOffset.bBusy OR FB_MBReadInputRegsSupPress.bBusy OR FB_MBReadInputRegsExhDamperPos.bBusy OR FB_MBReadInputRegsSupFlow.bBusy OR
	FB_MBReadInputRegsExhFlow.bBusy ;

END_FUNCTION_BLOCK

// oaksModbusLibrary/Vacon/fbVaconFO_1
//OAKS AB
//2023-02-22
//Funktionsblock för kommunikation via Modbus med VACON FO
FUNCTION_BLOCK fbVaconFO_1
VAR CONSTANT
	StartInputRegs_1	: INT :=2101;
	NrInputRegs_1 		: UINT := 11;

END_VAR
VAR_INPUT
	stAdd	: ST_ModbusTCP;
	nUnitID : UINT(1..254);
	bStart : BOOL;
	bSafe : BOOL;
	bReset : BOOL;
	rAnalogInput : REAL;
	tAlarmDelay : TIME := T#3S; // Larmfördröjning
	bAutoReset : BOOL := TRUE; // auto-reset utav driftfel
END_VAR
VAR_OUTPUT
	FAULT 	AT %M* 	: BOOL; //Kommunikationsfel frekvensomformare~wp:[alarmoptions]p:1
	PV8 	AT %M*	: STRING; //Modbus konfiguering~wp:
	V		AT %M* 	: BOOL; //Driftindikering~wp:[trendoptions]i:14400, t:1
	AL		AT %M* 	: BOOL; //Driftfel pump~wp:
	AL1		AT %M* 	: BOOL; //Summalarm pump~wp:
	PV		AT %M*  : REAL; //Hastighet~wp:[unit]%[format]0[trendoptions]i:300
	FO_OP 	AT %M*	: REAL; //Utsignal~wp:[unit]%[format]0[trendoptions]i:300
	FO_AL8 	AT %M* 	: BOOL; //Utsignal handställd~wp:[alarmoptions]p:3
	AL8		AT %M*	: BOOL; //Utsignal handställd~wp:[alarmoptions]p:3
	CMD		AT %M*  : BOOL; //Utsignal~wp:[trendoptions]i:14400, t:1
	
	bAlarmOutput : BOOL; // internvariabel larm , används för knytning till exempelvis aggregatsblock
END_VAR
VAR_IN_OUT
END_VAR
VAR
	iModbusLoop	: INT;	

	fbReadHoldingRegs_1 : FB_MBReadInputRegs;
	aInputRegs_1 : ARRAY[1..NrInputRegs_1] OF WORD;

	fbWriteControlWord : FB_MBWriteSingleReg;
	fbWriteSpeed	   : FB_MBWriteSingleReg;
	wValueToWrite : WORD;
	
	//Kommunikationsfel
	fbKommTof : tof; 
	fbKommTon : ton;

	//Övrigt
	Offset 				: INT :=-1;	
	bSekvensFlagga		: BOOL;
	sIP, sPort, sModbusID, sModbusLoop: STRING(255);
	bBusy_1x, bBusy_3x, bBusy_4x : BOOL;
	bError_1x, bError_3x, bError_4x : BOOL;

	bWriteActive : BOOL := TRUE;
	
	//Webport
//	V4 		AT %M*  : BOOL; //Standby bit (1=Standby)~wp:[trendoptions]i:300
//	PV5 	AT %M*  : BOOL; //Motionskörning~wp:[trendoptions]i:300
//	AL2 	AT %M*  : BOOL; //Övertemperatur (NTC)~wp:[trendoptions]i:300
	
	bAlarm : BOOL;
	fbAlarm1 : fbAlarm;
	
END_VAR
VAR_INPUT PERSISTENT
	M AT %M* : BOOL; //Handställning~wp:[trendoptions]i:14400, t:1
	MCMD AT %M* : BOOL; //Styrsignal handställning~wp:[trendoptions]i:14400, t:1
	FO_M  AT %M*: BOOL; //Handställning~wp:[trendoptions]i:14400, t:1
	FO_OPM AT %M*: REAL;//Värde handställning~wp:[unit]%[format]0
END_VAR

//Modbus konfiguering
	sIP := CONCAT (stAdd.sIPAddr, '');
	sPort := CONCAT ('<br>Port: ', UINT_TO_STRING(stAdd.nTCPPort));
	sModbusID := CONCAT('<br>ID: ', UINT_TO_STRING(nUnitID));
	sModbusLoop := CONCAT('<br>Loop: ', INT_TO_STRING(stAdd.iModbusLoop));
	iModbusLoop := stAdd.iModbusLoop;
	PV8 := CONCAT(CONCAT(CONCAT(sIP, sPort), sModbusID), sModbusLoop);

//Misc
IF (aInputRegs_1[11]=53) THEN 
	bReset := 1;
ELSE
	bReset := 0;
END_IF

FO_AL8 := FO_M;

IF FO_M THEN FO_OP := FO_OPM;
ELSE FO_OP := rAnalogInput;	
END_IF

IF M THEN CMD := MCMD;
ELSE CMD := bStart;	
END_IF

AL8		:= FO_M OR M;

	wValueToWrite.0 := CMD AND bSafe;
//	wValueToWrite.1 := ;
	wValueToWrite.2 := bReset;

//Sekvens	
	bSekvensFlagga := oaksGVL.aBModbusSekvens[iModbusLoop] = UINT_TO_INT(nUnitID);

//Read Input Status Registers
	bBusy_1x  := FALSE;
	bError_1x := FALSE;

//Reag Input Registers(Single)
	
//Read Input Registers (Multiple)
	fbReadHoldingRegs_1(sIPAddr:= stAdd.sIPAddr, nTCPPort:= stAdd.nTCPPort, nUnitID:= UINT_TO_BYTE(nUnitID), nQuantity:= NrInputRegs_1, nMBAddr:= INT_TO_WORD(StartInputRegs_1+Offset), cbLength:= SIZEOF(aInputRegs_1), pDestAddr:=ADR(aInputRegs_1), bExecute:= bSekvensFlagga, tTimeout:= T#3S, bBusy=> , bError=> , nErrId=> , cbRead=> );

	bBusy_3x  := fbReadHoldingRegs_1.bBusy;
	bError_3x := fbReadHoldingRegs_1.bError;
	
//Read Holding Regs

//Write Holding Registers (Single)
	fbWriteControlWord( sIPAddr:= stAdd.sIPAddr, nTCPPort:= stAdd.nTCPPort, nUnitID:= UINT_TO_BYTE(nUnitID), nMBAddr:= INT_TO_WORD(2001+Offset), nValue:= wValueToWrite, bExecute:= (bSekvensFlagga AND bWriteActive), tTimeout:= T#3S, bBusy=> , bError=> , nErrId=> );
	fbWriteSpeed( sIPAddr:= stAdd.sIPAddr, nTCPPort:= stAdd.nTCPPort, nUnitID:= UINT_TO_BYTE(nUnitID), nMBAddr:= INT_TO_WORD(2003+Offset), nValue:= REAL_TO_WORD(FO_OP*100), bExecute:= (bSekvensFlagga AND bWriteActive), tTimeout:= T#3S, bBusy=> , bError=> , nErrId=> );
	
	bBusy_4x :=  fbWriteControlWord.bBusy OR fbWriteSpeed.bBusy;
	bError_4x := fbWriteControlWord.bError OR fbWriteSpeed.bError;

//Convert values
PV		:=	WORD_TO_REAL(aInputRegs_1[3])/100;
V		:=	(aInputRegs_1[1].1 = 1);
AL1		:=	(aInputRegs_1[1].3 = 1);

//Write busy	
	oaksgvl.aBModbusBusyFlagga[iModbusLoop,nUnitID] := ( bBusy_1x OR bBusy_3x OR bBusy_4x );

//Communication error
	fbKommTof(IN:= 	bError_1x OR bError_3x OR bError_4x, PT:=T#3S , Q=> , ET=> );
	fbKommTon(IN:=fbKommTof.Q , PT:=T#1M , Q=> FAULT, ET=> );
	
//Driftfelslarm
	bAlarm := V XOR CMD;
	fbAlarm1(bInput:=bAlarm , tAlarmDelay:=tAlarmDelay , bAutoReset:=bAutoReset , bAlarmOutput=> AL);
	bAlarmOutput := AL;

END_FUNCTION_BLOCK

// oaksModbusLibrary/Wilo/fbWiloCif_If
(*
OAKS AB - Harri Seppänen
2020-05-12
Modbusblock för Wilo IF/CIF modul
*)
FUNCTION_BLOCK fbWiloCif_If EXTENDS fbMotorAo
VAR_INPUT
	sIPAddr : STRING := ''; 
	nTCPPort : UINT;
	nUnitID : UINT :=1;
	iModbusLoop : INT :=1; //Modbusslinga
			
END_VAR
VAR_OUTPUT
	PV AT %M*  : REAL; //Tryck~wp:[unit]kPa[format]0.0
	PV1 AT %M*  : REAL; //Flöde~wp:[unit]m³/h[format]0.0
	PV2 AT %M*  : REAL; //Effekt~wp:[unit]W[format]0
	PV3 AT %M*  : REAL; //Hastighet~wp:[unit]rpm[format]0
	PV4 AT %M*  : REAL; //Tryck (cm H₂O) ~wp:[unit]cm H₂O[format]0
	PV6 AT %M* : STRING;//Modbus konfiguering~wp:
	AL7 AT %M* : BOOL;//Kommunikationsfel~wp:
	
END_VAR
VAR
	uppdatering : BOOL := TRUE;
	offset : WORD;
	rTemp : REAL;
	iTemp : UINT;
	bSekvensFlagga : BOOL;
			
	FB_MBReadRegs_Input1_10: FB_MBReadInputRegs;
	ArrInput1_10 : ARRAY [1..10] OF WORD; //Holding
	//Kommunikationsfel
	fbKommTof : tof; 
	fbKommTon : fbAlarm;
	
	sIP: STRING(255);
	sPort: STRING(255);
	sModbusID: STRING(255);
	sModbusLoop: STRING(255);
	sTemp : STRING(255);
	
	fbReadWriteHoldingRegRealWriteSpeed : fbReadWriteHoldingRegReal;
	fbReadWriteHoldingRegRealWriteStart : fbReadWriteHoldingRegReal;
	
END_VAR

	SUPER^();
//General
	offset := 0;
//Sekvens
	bSekvensFlagga := oaksGVL.aBModbusSekvens[iModbusLoop] = UINT_TO_INT(nUnitID);
//Modbus konfiguering
	sIP := CONCAT (SIPAddr, '');
	sPort := CONCAT ('<br>Port: ', UINT_TO_STRING(nTCPPort)); 								
	sModbusID := CONCAT('<br>ID: ', UINT_TO_STRING(nUnitID));
	sModbusLoop := CONCAT('<br>Loop: ', INT_TO_STRING(iModbusLoop));	

	sTemp := sIP;
	sTemp := CONCAT(sTemp, sPort);
	sTemp := CONCAT(sTemp, sModbusID);
	sTemp := CONCAT(sTemp, sModbusLoop);
	
	PV6 := sTemp;
	
	///////////////
	//READ
	///////////////
	
	//Read Holding 0-10
	FB_MBReadRegs_Input1_10(
	sIPAddr:= sIpAddr, 
	nTCPPort:= INT_TO_UINT(nTCPPort), 
	nUnitID:= INT_TO_BYTE(nUnitID), 
	nQuantity:= 7, 
	nMBAddr:= 1 + offset, 
	cbLength:= SIZEOF(ArrInput1_10), 
	pDestAddr:= ADR(ArrInput1_10), 
	bExecute:= bSekvensFlagga, 
	tTimeout:= T#3S, 
	bBusy=> , 
	bError=> , 
	nErrId=> , 
	cbRead=> );
	
	PV4 := WORD_TO_REAL(ArrInput1_10[1]) * 10; //Pressure 	cm H2O
	PV := PV4 * 0.0980665; //Omvandling från cm H2O till kPa
	
	PV1 :=  WORD_TO_REAL(ArrInput1_10[2]) / 10; //Flow m³/h
	//WORD_TO_REAL(ArrHolding1_10[3]); //Energy Consumption kWh
	PV2 := WORD_TO_REAL(ArrInput1_10[4]); //Power input W
	//WORD_TO_REAL(ArrHolding1_10[5]); //Operation Time
	PV3 := WORD_TO_REAL(ArrInput1_10[7]); //Speed
	//WORD_TO_REAL(ArrHolding1_10[8]); //Temperature fluid @ device
	//WORD_TO_REAL(ArrHolding1_10[9]); //Operating Hours DP
	//WORD_TO_REAL(ArrHolding1_10[10]); //Control Function
	

	
	fbReadWriteHoldingRegRealWriteSpeed(
	sIPAddr:= sIpAddr, 
	nTCPPort:= INT_TO_UINT(nTCPPort), 
	nUnitID:= INT_TO_BYTE(nUnitID),  
	mBusAdr:= 1, 
	bEnable:= bSekvensFlagga, 
	tTimeout:= T#4S, 
	rReal:= FO_OP * 2, 
	uiFaktor:= 1, 
	bError=> , 
	bBusy=> , 
	bSuccess=> );
	
	IF CMD THEN
		fbReadWriteHoldingRegRealWriteStart.rReal := 9;
	ELSE
		fbReadWriteHoldingRegRealWriteStart.rReal := 0;
	END_IF
	
		
	fbReadWriteHoldingRegRealWriteStart(
	sIPAddr:= sIpAddr, 
	nTCPPort:= INT_TO_UINT(nTCPPort), 
	nUnitID:= INT_TO_BYTE(nUnitID), 
	mBusAdr:= 40, 
	bEnable:= bSekvensFlagga, 
	tTimeout:= T#4S, 
	uiFaktor:= 1, 
	bError=> , 
	bBusy=> , 
	bSuccess=> );
	
	//Communication error
	fbKommTof(IN:=FB_MBReadRegs_Input1_10.bError , PT:=T#20S , Q=> , ET=> );
	fbKommTon(bInput:=fbKommTof.Q , tAlarmDelay:=T#20M , bAutoReset:= , bAlarmOutput=> );
	AL7 :=fbKommTon.bAlarmOutput;
		
	//Write busy
	oaksgvl.aBModbusBusyFlagga[iModbusLoop,nUnitID] := FB_MBReadRegs_Input1_10.bBusy OR fbReadWriteHoldingRegRealWriteSpeed.bBusy OR fbReadWriteHoldingRegRealWriteStart.bBusy;

END_FUNCTION_BLOCK

// oaksModbusLibrary/Xylem/fbXylemEcocircXLplus
//OAKS AB
//2023-04-11 ver. b0.1
//Funktionsblock för modbus-TCP, Xylem ecocirc XLplus.

FUNCTION_BLOCK fbXylemEcocircXLplus
VAR_INPUT
	sIPAddr : STRING := ''; 
	nTCPPort : UINT;
	nUnitID : UINT :=1;
	iModbusLoop : INT :=1; //Modbusslinga	
END_VAR

VAR_OUTPUT
	P1 AT %M* : REAL;//Effekt~wp:[unit]W[format]0[trendoptions]i:300
	PV AT %M* : REAL;//Flöde~wp:[unit]l/s[format]0.0[trendoptions]i:300	
	RPM AT %M* : REAL;//Varvtal~wp:[unit]RPM[format]0[trendoptions]i:300
	PV1 AT %M* : REAL;//Temperatur vatten~wp:[unit]°C[format]0.0[trendoptions]i:300
	I1 AT %M* : REAL;//Ström~wp:[unit]A[format]0.00[trendoptions]i:300
	V3 AT %M* : BOOL;//Start/Stopp~wp:[trendoptions]i:14400, t:1
	PV8 AT %M* : STRING;//Modbus konfiguering~wp:
	FAULT AT %M* : BOOL;//Kommunikationsfel~wp:[alarmoptions]p:2
END_VAR
VAR
	offset : WORD;;
	bSekvensFlagga : BOOL;
			
	FB_MBReadRegs_ArrHolding1 : FB_MBReadRegs;
	FB_MBReadRegs_StatusBits1 : FB_MBReadRegs;
	ArrHolding1 : ARRAY [0..10] OF WORD; //Read Holding Hex 200-20A / Dec 512-522
	
	wPower : WORD;
	wFlow : WORD;
	wSpeed  : WORD;
	wWaterTemperature : WORD;
	wCurrent : WORD;
	wStatusBits : WORD;
	
	//Kommunikationsfel
	fbKommTof : tof; 
	fbKommTon : fbAlarm;
	
	sIP: STRING(255);
	sPort: STRING(255);
	sModbusID: STRING(255);
	sModbusLoop: STRING(255);
	sTemp : STRING(255);
	
END_VAR

//General
	offset := 0;
//Sekvens	
	bSekvensFlagga := oaksGVL.aBModbusSekvens[iModbusLoop] = UINT_TO_INT(nUnitID);
//Modbus konfiguering
	sIP := CONCAT (SIPAddr, '');
	sPort := CONCAT ('<br>Port: ', UINT_TO_STRING(nTCPPort)); 								
	sModbusID := CONCAT('<br>ID: ', UINT_TO_STRING(nUnitID));
	sModbusLoop := CONCAT('<br>Loop: ', INT_TO_STRING(iModbusLoop));	

	sTemp := sIP;
	sTemp := CONCAT(sTemp, sPort);
	sTemp := CONCAT(sTemp, sModbusID);
	sTemp := CONCAT(sTemp, sModbusLoop);
	
	PV8 := sTemp;

///////////////		
//READ
///////////////		
	
	//Read Holding Hex 200-20A / Dec 512-522
	FB_MBReadRegs_ArrHolding1(
	sIPAddr:= sIpAddr, 
	nTCPPort:= INT_TO_UINT(nTCPPort), 
	nUnitID:= INT_TO_BYTE(nUnitID), 
	nQuantity:= 11, 
	nMBAddr:= 512 + offset, 
	cbLength:= SIZEOF(ArrHolding1), 
	pDestAddr:= ADR(ArrHolding1), 
	bExecute:= bSekvensFlagga, 
	tTimeout:= T#3S, 
	bBusy=> , 
	bError=> , 
	nErrId=> , 
	cbRead=> );
	
	//Values
	wPower := ArrHolding1[0]; //"INPUT POWER"
	P1 := WORD_TO_REAL(wPower);
	wFlow := ArrHolding1[2]; //"FLOW"
	PV := WORD_TO_REAL(wFlow)*0.1;
	wSpeed := ArrHolding1[3]; //"SPEED"
	RPM := WORD_TO_REAL(wSpeed);
	wWaterTemperature := ArrHolding1[4]; //"WATER TEMPERATURE"
	PV1 := WORD_TO_REAL(wWaterTemperature)*0.1;
	wCurrent := ArrHolding1[10]; //"QUADRATURE CURRENT"
	I1 := WORD_TO_REAL(wCurrent)*0.01;
	
	//Read Holding Hex 20B / Dec 523
	FB_MBReadRegs_StatusBits1(
	sIPAddr:= sIpAddr, 
	nTCPPort:= INT_TO_UINT(nTCPPort), 
	nUnitID:= INT_TO_BYTE(nUnitID), 
	nQuantity:= 1, 
	nMBAddr:= 523 + offset, 
	cbLength:= SIZEOF(wStatusBits), 
	pDestAddr:= ADR(wStatusBits), 
	bExecute:= bSekvensFlagga, 
	tTimeout:= T#3S, 
	bBusy=> , 
	bError=> , 
	nErrId=> , 
	cbRead=> );	
	
	V3 := wStatusBits.2; //"BIT FIELDS STATUS I/O - START/STOP SIGNAL STATUS"
	
//Communication error
	fbKommTof(IN:=FB_MBReadRegs_ArrHolding1.bError , PT:=T#20S , Q=> , ET=> );
	fbKommTon(bInput:=fbKommTof.Q , tAlarmDelay:=T#20M , bAutoReset:= , bAlarmOutput=> );
	FAULT :=fbKommTon.bAlarmOutput;
		
//Write busy	
	oaksgvl.aBModbusBusyFlagga[iModbusLoop,nUnitID] := FB_MBReadRegs_Arrholding1.bBusy;

END_FUNCTION_BLOCK

// oaksModbusLibrary/Xylem/fbXylemHydrovarHVL
//OAKS AB
//2023-03-13 ver. b0.1
//Funktionsblock för modbus-TCP, Xylem Hydrovar HVL 2.015 - 4.220, Version SW 2.10 och 2.20.

FUNCTION_BLOCK fbXylemHydrovarHVL
VAR_INPUT
	sIPAddr : STRING := ''; 
	nTCPPort : UINT;
	nUnitID : UINT :=1;
	iModbusLoop : INT :=1; //Modbusslinga	
END_VAR

VAR_OUTPUT
	V3 AT %M* : BOOL;//Start/Stopp~wp:[trendoptions]i:14400, t:1
	PV AT %M* : REAL;//Aktuellt tryck~wp:[unit]Bar[format]0.00[trendoptions]i:300
	F AT %M* : REAL;//Frekvens~wp:[unit]Hz[format]0.0[trendoptions]i:300
	U1 AT %M* : REAL;//Spänning~wp:[unit]V[format]0[trendoptions]i:300
	I1 AT %M* : REAL;//Ström av max~wp:[unit]%[format]0.0[trendoptions]i:300
	E1 AT %M* : REAL;//Energi~wp:[unit]kWh[format]0[trendoptions]i:300	
	PV8 AT %M* : STRING;//Modbus konfiguering~wp:
	FAULT AT %M* : BOOL;//Kommunikationsfel~wp:[alarmoptions]p:2
END_VAR
VAR
	offset : WORD;
	iTemp1 : UINT;
	iTemp2 : UINT;
	bSekvensFlagga : BOOL;
			
	FB_MBReadRegs_ArrHolding1: FB_MBReadRegs;
	ArrHolding1 : ARRAY [0..3] OF WORD; //Read Holding Dec 49-51
	FB_MBReadRegs_ArrHolding2: FB_MBReadRegs;
	ArrHolding2 : ARRAY [0..1] OF WORD; //Read Holding Dec 109-110
	FB_MBReadRegs_ArrHolding3: FB_MBReadRegs;
	ArrHolding3 : ARRAY [0..1] OF WORD; //Read Holding Dec 135-136
	
	wStoppStart : WORD;
	wActualValue : WORD;
	wOutputValue : WORD;
	wKwhCounter1 : WORD;
	wKwhCounter2 : WORD;
	iKwhCounter : UDINT;
	wCurrInverter : WORD;
	wVoltInverter : WORD;
	
	//Kommunikationsfel
	fbKommTof : tof; 
	fbKommTon : fbAlarm;
	
	sIP: STRING(255);
	sPort: STRING(255);
	sModbusID: STRING(255);
	sModbusLoop: STRING(255);
	sTemp : STRING(255);
	
END_VAR

//General
	offset := 0;
//Sekvens	
	bSekvensFlagga := oaksGVL.aBModbusSekvens[iModbusLoop] = UINT_TO_INT(nUnitID);
//Modbus konfiguering
	sIP := CONCAT (SIPAddr, '');
	sPort := CONCAT ('<br>Port: ', UINT_TO_STRING(nTCPPort)); 								
	sModbusID := CONCAT('<br>ID: ', UINT_TO_STRING(nUnitID));
	sModbusLoop := CONCAT('<br>Loop: ', INT_TO_STRING(iModbusLoop));	

	sTemp := sIP;
	sTemp := CONCAT(sTemp, sPort);
	sTemp := CONCAT(sTemp, sModbusID);
	sTemp := CONCAT(sTemp, sModbusLoop);
	
	PV8 := sTemp;

///////////////		
//READ
///////////////		
	
	//Read Holding Dec 49-51
	FB_MBReadRegs_ArrHolding1(
	sIPAddr:= sIpAddr, 
	nTCPPort:= INT_TO_UINT(nTCPPort), 
	nUnitID:= INT_TO_BYTE(nUnitID), 
	nQuantity:= 3, 
	nMBAddr:= 49 + offset, 
	cbLength:= SIZEOF(ArrHolding1), 
	pDestAddr:= ADR(ArrHolding1), 
	bExecute:= bSekvensFlagga, 
	tTimeout:= T#3S, 
	bBusy=> , 
	bError=> , 
	nErrId=> , 
	cbRead=> );
	
	//Values
	wStoppStart := ArrHolding1[0]; //"STOP/START"
	V3 := WORD_TO_BOOL(wStoppStart);
	wActualValue := ArrHolding1[1]; //"ACTUAL VALUE"
	PV := WORD_TO_REAL(wActualValue)*0.01;
	wOutputValue := ArrHolding1[2]; //"OUTPUT FREQ."
	F := WORD_TO_REAL(wOutputValue)*0.1;

	//Read Holding Dec 109-110
	FB_MBReadRegs_ArrHolding2(
	sIPAddr:= sIpAddr, 
	nTCPPort:= INT_TO_UINT(nTCPPort), 
	nUnitID:= INT_TO_BYTE(nUnitID), 
	nQuantity:= 2, 
	nMBAddr:= 109 + offset, 
	cbLength:= SIZEOF(ArrHolding2), 
	pDestAddr:= ADR(ArrHolding2), 
	bExecute:= bSekvensFlagga, 
	tTimeout:= T#3S, 
	bBusy=> , 
	bError=> , 
	nErrId=> , 
	cbRead=> );

	//Values
	wKwhCounter1 := ArrHolding2[0]; //"KWH COUNTER"
	iTemp1 := wKwhCounter1;
	wKwhCounter2 := ArrHolding2[1]; //"KWH COUNTER"
	iTemp2 := WORD_TO_UINT(wKwhCounter2);
	iKwhCounter := ((iTemp1*65536) + iTemp2);
	E1 := UDINT_TO_REAL(iKwhCounter);

	//Read Holding Dec 135-136
	FB_MBReadRegs_ArrHolding3(
	sIPAddr:= sIpAddr, 
	nTCPPort:= INT_TO_UINT(nTCPPort), 
	nUnitID:= INT_TO_BYTE(nUnitID), 
	nQuantity:= 2, 
	nMBAddr:= 135 + offset, 
	cbLength:= SIZEOF(ArrHolding3), 
	pDestAddr:= ADR(ArrHolding3), 
	bExecute:= bSekvensFlagga, 
	tTimeout:= T#3S, 
	bBusy=> , 
	bError=> , 
	nErrId=> , 
	cbRead=> );

	//Values
	wCurrInverter := ArrHolding3[0]; //"CURR.INVERTER"
	I1 := WORD_TO_REAL(wCurrInverter)*0.1;
	wVoltInverter := ArrHolding3[1]; //"VOLT.INVERTER"
	U1 := WORD_TO_REAL(wVoltInverter);	
	
//Communication error
	fbKommTof(IN:=FB_MBReadRegs_ArrHolding1.bError , PT:=T#20S , Q=> , ET=> );
	fbKommTon(bInput:=fbKommTof.Q , tAlarmDelay:=T#20M , bAutoReset:= , bAlarmOutput=> );
	FAULT :=fbKommTon.bAlarmOutput;
		
//Write busy	
	oaksgvl.aBModbusBusyFlagga[iModbusLoop,nUnitID] := FB_MBReadRegs_Arrholding1.bBusy;

END_FUNCTION_BLOCK
